// TIA Portal project "PLCSim Advanced 4.0" (V16)

(* hardware
DEVICE "PC-System_1"  SIMATIC PC station
   slot 0: "SIMATIC PC station"  Rail  SIMATIC PC-Station  V1.0
      slot 125: "Stationmanager"  Station_Manager  V6.0.4
   slot 1: "HMI_RT_1"  WinCC RT Professional  6AV2 105-0xxxx-xxxx  16.0.0.0
DEVICE "S71500/ET200MP station_1"  S7-1500 station
   slot 0: "Rail_0"  Rack  6ES7 590-1***0-0AA0
   slot 1: "PLC_1"  CPU 1513-1 PN  6ES7 513-1AL02-0AB0  V2.8
      slot 3: "CPU display_1"  6ES7591-1AA00-0AA0
      slot 32768: "PROFINET interface_1"  X1
         slot 32769: "Port_1"  X1 P1
         slot 32770: "Port_2"  X1 P2
      slot 34817: "Virtual CP interface port_1"  Virtual CP interface port  Virtual CP interface port
*)

// ===== PLC "PLC_1"  CPU 1513-1 PN =====

VAR_GLOBAL   // PLC tag table "Default tag table"
   "START" AT %M0.0 : Bool;
   "STOP" AT %M0.1 : Bool;
   "MOTOR" AT %M0.2 : Bool;
END_VAR

ORGANIZATION_BLOCK "Main"   // OB1, LAD, ProgramCycle
TITLE = "Main Program Sweep (Cycle)"
{ S7_Optimized_Access := 'TRUE' }
VERSION : 0.1
   VAR_INPUT
      Initial_Call : Bool;   // Initial call of this OB
      Remanence : Bool;   // =True, if remanent data are available
   END_VAR
BEGIN

REGION Network 1
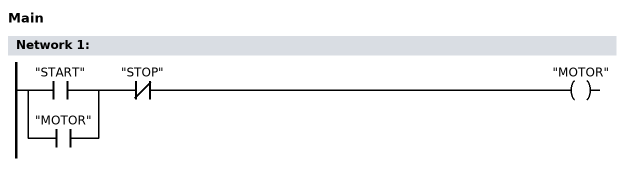
   RUNG wire#powerrail
      Contact( "START" )
      wire#w1
      I_Contact( "STOP" )
      Coil( "MOTOR" )
   END_RUNG
   RUNG wire#powerrail
      Contact( "MOTOR" )
   END_RUNG wire#w1
   // the same network as SCL:
   "MOTOR" := ("START" OR "MOTOR") AND NOT "STOP";
END_REGION
END_ORGANIZATION_BLOCK

(* ===== HMI "HMI_RT_1" =====
system functions are stored by id; their names below are inferred from use
connection "Connection_1": S71200_TCP_IP, SCADA_S7_1500_OMS

HMI tags "Default tag table"
   "START" : Bool AT %M0.0, 500 ms
   "STOP" : Bool AT %M0.1, 500 ms
   "MOTOR" : Bool AT %M0.2, 500 ms

screen "Screen_1" 1024x768
   Button "Button_1" at 143,131 size 121x34; TextOff 'Start'
      on PressLeft: SetBit("START")
      on ReleaseLeft: ResetBit("START")
   Button "Button_2" at 145,178 size 121x34; TextOff 'Stop'
      on PressLeft: SetBit("STOP")
      on ReleaseLeft: ResetBit("STOP")
   Circle "Circle_1" at 297,140 size 48x48
      Appearance <- "MOTOR"
*)